{attribute 'qualified_only'}
{attribute 'strict'}
{attribute 'to_string'}
TYPE E_MotionAxisPowerMode :
(
    enum_member := 0
);
END_TYPE

(* stored: Version 1.1.0.1
   DUT E_MotionAxisPowerMode: Id {17b79f2a-9dfd-44a5-a205-1783fa922e2c} *)
